// TwinCAT 3 PLC project PLC1
// ProgramVersion: 3.1.4023.0
// libraries:
//   Tc2_Standard, * (Beckhoff Automation GmbH)
//   Tc2_System, * (Beckhoff Automation GmbH)
//   Tc3_Module, * (Beckhoff Automation GmbH)
// project tree:
//   DUTs/ ST_DUT1.TcDUT, ST_ELDUTTO2.TcDUT
//   / PlcTask.TcTTO
//   POUs/ MAIN.TcPOU
// real-time tasks:
//   TASK PlcTask: cycle T#10ms, priority 20, ADS port 350

CONFIGURATION PLC1
    RESOURCE PLC ON TwinCAT3
        TASK PlcTask(INTERVAL := T#10ms, PRIORITY := 20);
        PROGRAM MAIN WITH PlcTask : MAIN;
    END_RESOURCE
END_CONFIGURATION

// ---- DUTs/ST_DUT1.TcDUT
TYPE ST_DUT1 :
STRUCT
	blol:BOOL;
END_STRUCT
END_TYPE

// ---- DUTs/ST_ELDUTTO2.TcDUT
TYPE ST_ELDUTTO2 :
STRUCT
	bDuttos:BOOL;
END_STRUCT
END_TYPE

// ---- POUs/MAIN.TcPOU
PROGRAM MAIN
VAR
END_VAR

END_PROGRAM
